VAR_GLOBAL
	ProcessTimers : ARRAY [0..20] OF TON;
END_VAR

(* stored: Version 1.1.0.1
   GVL M1_AUX: Id {6bbe7c60-acb3-44ce-8c7b-c7d66b25a177} *)
